Fanuc TP program (LS listing): KFKEEP.LS

/PROG  KFKEEP
/ATTR
OWNER		= MNEDITOR;
COMMENT		= "KAREL file left open";
PROG_SIZE	= 0;
CREATE		= DATE 26-01-01  TIME 00:00:00;
MODIFIED	= DATE 26-01-01  TIME 00:00:00;
FILE_NAME	= ;
VERSION		= 0;
LINE_COUNT	= 2;
MEMORY_SIZE	= 0;
PROTECT		= READ_WRITE;
TCD:  STACK_SIZE	= 0,
      TASK_PRIORITY	= 50,
      TIME_SLICE	= 0,
      BUSY_LAMP_OFF	= 0,
      ABORT_REQUEST	= 0,
      PAUSE_REQUEST	= 0;
DEFAULT_GROUP	= 1,*,*,*,*;
CONTROL_CODE	= 00000000 00000000;
/MN
   1:  CALL CA_FILE(1,95,1,'UD1:','kfkeep.txt') ;
   2:  CALL CA_FILE(2,95,1,'a') ;
/POS
/END
